FUNCTION_BLOCK FB_StationUnloadElevator
VAR_INPUT
	Enable:				BOOL;
	System:				REFERENCE TO ST_System;
	Station:			REFERENCE TO ST_SystemStation;
	Error:				REFERENCE TO ST_Error;
	Setting:			REFERENCE TO ST_Setting;
	Recipe:				REFERENCE TO ST_Recipe;	
	Parameter:			REFERENCE TO ST_StationUnloadElevator;
END_VAR
VAR_OUTPUT
END_VAR
VAR
	_stHandshake: ST_StationUnloadElevatorHandshake;
END_VAR

A_Auto();
A_Home();

ACTION A_Auto:
CASE Station.iStepNow OF
	1000:
		Station.arrInfo[E_Language.Chinese]:="初始化完成 等待启动";
		IF Enable THEN
			Station.iStepNext:=1101;
		END_IF
	1101:
		Station.arrInfo[E_Language.Chinese]:="判断是否有料";
		IF NOT Parameter.bFrockElevator1NoneCheck THEN
			Station.iStepNext:=1201;
		END_IF
	1201:
		Station.arrInfo[E_Language.Chinese]:="等待拆解站请求放料";
		IF Parameter.stHandshake.bRequestElevator THEN
			Parameter.stHandshake.bResponseDismantling_E:=TRUE;
			Station.iStepNext:=1301;
		END_IF
	1301:
		Station.arrInfo[E_Language.Chinese]:="等待产品到位";
		IF Parameter.bFrockElevator1NoneCheck THEN
			Station.iStepNext:=1351;
		END_IF
	1351:
		Station.arrInfo[E_Language.Chinese]:="等待复位放料请求";
		IF NOT Parameter.stHandshake.bRequestElevator THEN
			Parameter.stHandshake.bResponseDismantling_E:=FALSE;
			Station.iStepNext:=1401;
		END_IF
	1401:
		Station.arrInfo[E_Language.Chinese]:="锁紧工装";
		IF Parameter.fbFrockRotateDown.M_HomeRequest() THEN
			Station.iStepNext:=1501;
		END_IF
	1501:
		Station.arrInfo[E_Language.Chinese]:="提升气缸上升";
		IF Parameter.fbFrockElevator.M_WorkRequest() THEN
			Station.iStepNext:=1601;
		END_IF
	1601:
		Station.arrInfo[E_Language.Chinese]:="松开工装";
		IF Parameter.fbFrockRotateDown.M_WorkRequest() THEN
			Station.iStepNext:= SEL(Parameter.bManualUnload,1701,1801);
		END_IF
	1701:
		Station.arrInfo[E_Language.Chinese]:="向下线体请求放料";
		Parameter.stHandshake.bRequestUnline:=TRUE;
		IF Parameter.stHandshake.bResponseElevator THEN
			Station.iStepNext:=1801;
		END_IF
	1801:
		Station.arrInfo[E_Language.Chinese]:="拨料气缸伸出";
		IF Parameter.fbFrockPush.M_WorkRequest() THEN
			Station.iStepNext:=1901;
		END_IF
	1901:
		Station.arrInfo[E_Language.Chinese]:="拨料气缸缩回";
		IF Parameter.fbFrockPush.M_HomeRequest() THEN
			Station.iStepNext:=SEL(Parameter.bManualUnload,2001,2101);
		END_IF
	2001:
		Station.arrInfo[E_Language.Chinese]:="复位放料请求";
		Parameter.stHandshake.bRequestUnline:=FALSE;
		IF NOT Parameter.stHandshake.bResponseElevator THEN
			Station.iStepNext:=2101;
		END_IF
	2101:
		Station.arrInfo[E_Language.Chinese]:="旋转压紧气缸缩回";
		IF Parameter.fbFrockRotateDown.M_HomeRequest() THEN
			Station.iStepNext:=2201;
		END_IF
	2201:
		Station.arrInfo[E_Language.Chinese]:="提升气缸下降";
		IF Parameter.fbFrockElevator.M_HomeRequest() THEN
			Station.iStepNext:=2301;
		END_IF
	2301:
		Station.arrInfo[E_Language.Chinese]:="旋转压紧气缸伸出";
		IF Parameter.fbFrockRotateDown.M_WorkRequest() THEN
			Station.iStepNext:=1101;
		END_IF
END_CASE
END_ACTION

ACTION A_Home:
CASE Station.iStepNow OF
	0:
		Station.arrInfo[E_Language.Chinese]:="等待初始化";
		Parameter.stHandshake:=_stHandshake;
		Station.iStepNext:=SEL(Enable,1000,100);
	100:
		Station.arrInfo[E_Language.Chinese]:="拨料气缸复位";
		IF Parameter.fbFrockPush.M_HomeRequest() THEN
			Station.iStepNext:=200;
		END_IF
	200:
		Station.arrInfo[E_Language.Chinese]:="旋转压紧气缸缩回";
		IF Parameter.fbFrockRotateDown.M_HomeRequest() THEN
			Station.iStepNext:=300;
		END_IF
	300:
		Station.arrInfo[E_Language.Chinese]:="提升气缸下降";
		IF Parameter.fbFrockElevator.M_HomeRequest() THEN
			Station.iStepNext:=400;
		END_IF
	400:
		Station.arrInfo[E_Language.Chinese]:="旋转压紧气缸伸出";
		IF Parameter.fbFrockRotateDown.M_WorkRequest() THEN
			Station.iStepNext:=1000;
		END_IF
END_CASE
END_ACTION

END_FUNCTION_BLOCK

(* stored: Version 1.1.0.1, ProductVersion 3.1.4024.3
   POU FB_StationUnloadElevator: Id {210b3d4c-3b29-4224-b2f1-f2015b60c563}, SpecialFunc None
   Action A_Auto: Id {a4d99731-efeb-4b35-a297-2da5d14c9920}
   Action A_Home: Id {16aa9363-a193-455f-9c58-c26dec971fd7} *)
